KUKA KRL program: Rack_Azul_Abrir_PLC.src, Rack_Azul_Abrir_PLC.dat

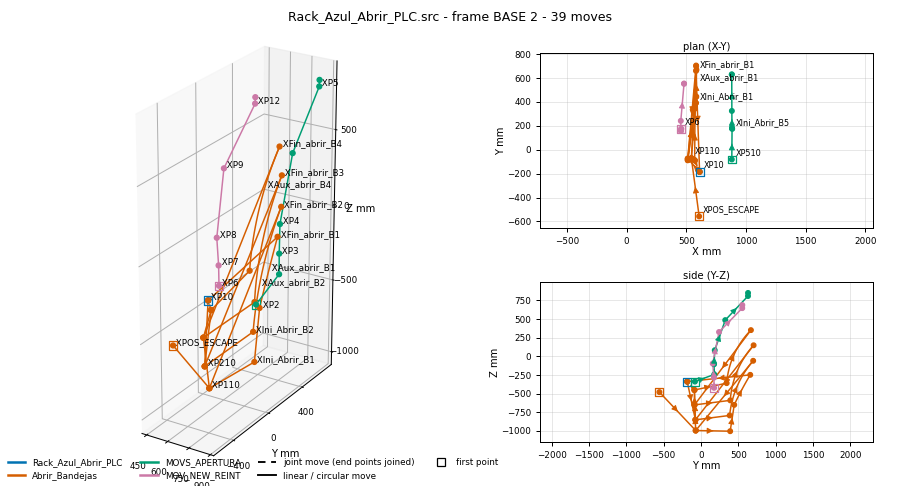
[picture p0: tool path of Rack_Azul_Abrir_PLC.src in frame BASE 2, 39 of 50 moves have a stored position in this frame; points joined in program order, loops and branches not executed]
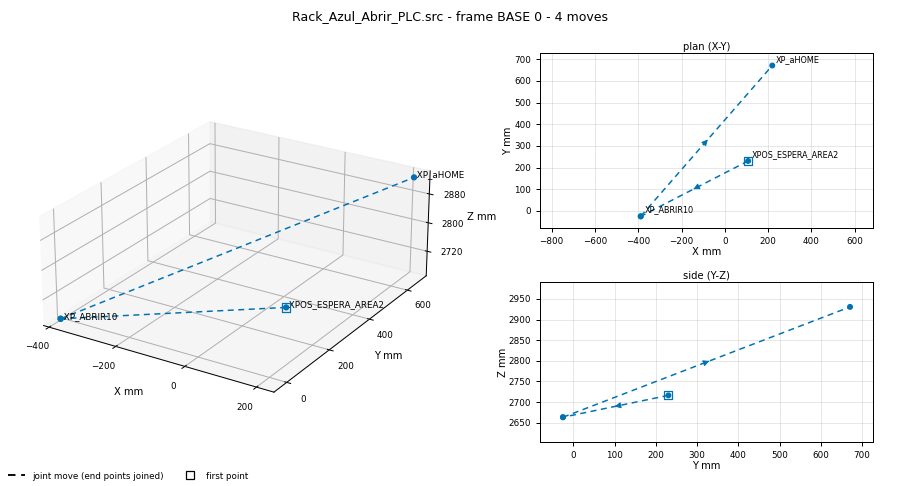
[picture p1: tool path of Rack_Azul_Abrir_PLC.src in frame BASE 0, 4 of 50 moves have a stored position in this frame; points joined in program order, loops and branches not executed]
--- Rack_Azul_Abrir_PLC.src ---
&ACCESS RVO1
&REL 29
&COMMENT ABRIR BAND RACK AZUL
&PARAM EDITMASK = *
&PARAM TEMPLATE = C:\KRC\Roboter\Template\vorgabe
&PARAM DISKPATH = KRC:\R1\Program\MAFELEC
DEF Rack_Azul_Abrir_PLC( )
;FOLD INI;%{PE}
  ;FOLD BASISTECH INI
    GLOBAL INTERRUPT DECL 3 WHEN $STOPMESS==TRUE DO IR_STOPM ( )
    INTERRUPT ON 3
    BAS (#INITMOV,0 )
  ;ENDFOLD (BASISTECH INI)
;FOLD SPOTTECH INI
USERSPOT(#INIT)
;ENDFOLD (SPOTTECH INI)
;FOLD GRIPPERTECH INI
USER_GRP(0,DUMMY,DUMMY,GDEFAULT)
;ENDFOLD (GRIPPERTECH INI)
  ;FOLD USER INI
    ;Make your modifications here
INTERRUPT DECL 21 WHEN I_Rack2_S1 DO Paro()
INTERRUPT DECL 22 WHEN I_Rack2_S2 DO Paro()
INTERRUPT DECL 23 WHEN I_Rack2_S3 DO Paro()
INTERRUPT DECL 24 WHEN I_Rack2_S4 DO Paro()
INTERRUPT DECL 25 WHEN I_Rack2_S5 DO Paro()
INTERRUPT DECL 81 WHEN I_121R1S501 DO STOP_PUSH ()
INTERRUPT DECL 82 WHEN I_121R1S502 DO STOP_PUSH ()
O_TYPE_INFO=0

  ;ENDFOLD (USER INI)
;ENDFOLD (INI)
;################################################
; PROYECTO: MAFELEC PLANTA DE BATERIAS
; ROBOT: 121_R1
; PROGRAMA: APERTURA DE BANDEJAS EN RACK AZUL
; CREADO POR: Su Majestad Felipe VI(zaisor robotics)
; FECHA: 23-NOVIEMBRE-2022
; MODIFICADO POR:
; FECHA MODIFICACION: 18-ENERO-2023
;################################################

Empujador(1,"A",FALSE)
Empujador(2,"R",FALSE)

; POSICION DE ESPERA ENTRADA RACK 2 (AZUL)
;FOLD PTP POS_ESPERA_AREA2 Vel=100 % H Tool[9]:T_Gripper1_Vacio Base[0];%{PE}%R 8.3.48,%MKUKATPBASIS,%CMOVE,%VPTP,%P 1:PTP, 2:POS_ESPERA_AREA2, 3:, 5:100, 7:H
$BWDSTART=FALSE
PDAT_ACT=PH
FDAT_ACT=FPOS_ESPERA_AREA2
BAS(#PTP_PARAMS,100)
PTP XPOS_ESPERA_AREA2
;ENDFOLD

$TIMER[6]=0
$TIMER_STOP[6]=FALSE

;ESPERA AREA 2
WAIT FOR I_ARDY_2
O_AREL_2=FALSE

WAIT FOR I_121R1S1000==FALSE
;INTERRUPT ON 81
;INTERRUPT ON 91

;FOLD PTP P_ABRIR10 CONT Vel=100 % H Tool[9]:T_Gripper1_Vacio Base[0];%{PE}%R 8.3.48,%MKUKATPBASIS,%CMOVE,%VPTP,%P 1:PTP, 2:P_ABRIR10, 3:C_DIS, 5:100, 7:H
$BWDSTART=FALSE
PDAT_ACT=PH
FDAT_ACT=FP_ABRIR10
BAS(#PTP_PARAMS,100)
PTP XP_ABRIR10 C_DIS
;ENDFOLD

;FOLD PTP P10 Vel=100 % H Tool[1]:T_PUSH1 Base[2]:Rack_Azul;%{PE}%R 8.3.48,%MKUKATPBASIS,%CMOVE,%VPTP,%P 1:PTP, 2:P10, 3:, 5:100, 7:H
$BWDSTART=FALSE
PDAT_ACT=PH
FDAT_ACT=FP10
BAS(#PTP_PARAMS,100)
PTP XP10
;ENDFOLD

Empujador(1,"A",TRUE)
Empujador(2,"R",TRUE)

Repite:
Abrir_Bandejas ()

IF INTERRUPT_ACTV THEN
PTP $POS_ACT
GOTO Repite
ENDIF

;FOLD PTP P10 Vel=100 % H Tool[1]:T_PUSH1 Base[2]:Rack_Azul;%{PE}%R 8.3.48,%MKUKATPBASIS,%CMOVE,%VPTP,%P 1:PTP, 2:P10, 3:, 5:100, 7:H
$BWDSTART=FALSE
PDAT_ACT=PH
FDAT_ACT=FP10
BAS(#PTP_PARAMS,100)
PTP XP10
;ENDFOLD

; TRABAJO REALIZADO
O_JRDY_2=TRUE

IF FINALIZA_AZUL==FALSE THEN
O_TYPE_RQ=TRUE
WAIT FOR I_TYPE_INFO==1
ENDIF

O_TYPE_RQ=FALSE

Empujador(1,"R",FALSE)
Empujador(2,"R",FALSE)

; POSICION DE SALIDA RACK 2 (AZUL)
;FOLD PTP POS_AREA2_LIBRE Vel=100 % H Tool[9]:T_Gripper1_Vacio Base[0];%{PE}%R 8.3.48,%MKUKATPBASIS,%CMOVE,%VPTP,%P 1:PTP, 2:POS_AREA2_LIBRE, 3:, 5:100, 7:H
$BWDSTART=FALSE
PDAT_ACT=PH
FDAT_ACT=FPOS_AREA2_LIBRE
BAS(#PTP_PARAMS,100)
PTP XPOS_AREA2_LIBRE
;ENDFOLD
O_AREL_2=TRUE
Empujador(1,"R",TRUE)
Empujador(2,"R",TRUE)

;FOLD PTP P_aHOME CONT Vel=100 % H Tool[9]:T_Gripper1_Vacio Base[0];%{PE}%R 8.3.48,%MKUKATPBASIS,%CMOVE,%VPTP,%P 1:PTP, 2:P_aHOME, 3:C_DIS, 5:100, 7:H
$BWDSTART=FALSE
PDAT_ACT=PH
FDAT_ACT=FP_aHOME
BAS(#PTP_PARAMS,100)
PTP XP_aHOME C_DIS
;ENDFOLD
INTERRUPT OFF 81
INTERRUPT OFF 82

END
DEF Abrir_Bandejas ()

INI_BUCLE:
PTP $POS_ACT
INTERRUPT_ACTV=FALSE

INTERRUPT DECL 86 WHEN I_121R1S501 DO INT_6970 ()
INTERRUPT DECL 87 WHEN I_121R1S502 DO INT_6970 ()
INTERRUPT DECL 88 WHEN I_121R1S501 DO STOP_INT_REINT()
INTERRUPT DECL 89 WHEN I_121R1S502 DO STOP_INT_REINT()
INTERRUPT OFF 86
INTERRUPT OFF 87
INTERRUPT OFF 88
INTERRUPT OFF 89

IF TORQ_HAB THEN
;FOLD TORQMON SetLimits Axis1: 50 % Axis2: 50 % Axis3: 50 % Axis4: 50 % Axis5: 50 % Axis6: 50 %;%{PE}%R 8.3.48,%MKUKATPBASIS,%CTQ_MON,%VTQ_LIMITS,%P 2:TQ_LIMITS, 4:50, 7:50, 10:50, 13:50, 16:50, 19:50
SET_TQ_VALUES (50,50,50,50,50,50)
;ENDFOLD
ENDIF

O_TYPE_RQ=FALSE
WAIT FOR I_TYPE_INFO==0

O_TYPE_RQ=TRUE
WAIT FOR (I_TYPE_INFO > 0) AND (I_TYPE_INFO < 26)
RA_Bandeja_Nr=I_TYPE_INFO
O_TYPE_INFO=I_TYPE_INFO

;PETICION APERTURA BANDEJAS EN RACK 2 (AZUL)
SWITCH RA_Bandeja_Nr ;

CASE 1
O_TYPE_RQ=FALSE
FINALIZA_AZUL=TRUE
;FOLD LIN POS_ESCAPE Vel=1 m/s H Tool[2]:T_PUSH2 Base[2]:Rack_Azul;%{PE}%R 8.3.48,%MKUKATPBASIS,%CMOVE,%VLIN,%P 1:LIN, 2:POS_ESCAPE, 3:, 5:1, 7:H
$BWDSTART=FALSE
LDAT_ACT=LH
FDAT_ACT=FPOS_ESCAPE
BAS(#CP_PARAMS,1)
LIN XPOS_ESCAPE
;ENDFOLD
GOTO FIN

CASE 21
; TRABAJO REALIZADO
O_JRDY_5=FALSE

O_TYPE_RQ=FALSE
FINALIZA_AZUL=FALSE
;FOLD ACTIVA BUSQUEDA APERTURA BANDEJA 1
INTERRUPT ON 21
OLD_OVPRO=$OV_PRO
$ADVANCE=0
;ENDFOLD
WAIT FOR I_Rack2_S2==TRUE
WAIT FOR I_Rack2_S1==FALSE

WAIT FOR I_RackAzul_Pin2A
WAIT FOR I_RackAzul_Pin1B

;FOLD LIN P110 CONT Vel=1 m/s M Tool[1]:T_PUSH1 Base[2]:Rack_Azul;%{PE}%R 8.3.48,%MKUKATPBASIS,%CMOVE,%VLIN,%P 1:LIN, 2:P110, 3:C_DIS C_DIS, 5:1, 7:M
$BWDSTART=FALSE
LDAT_ACT=LM
FDAT_ACT=FP110
BAS(#CP_PARAMS,1)
LIN XP110 C_DIS C_DIS
;ENDFOLD

;FOLD LIN Ini_Abrir_B1 Vel=1 m/s M Tool[1]:T_PUSH1 Base[2]:Rack_Azul;%{PE}%R 8.3.48,%MKUKATPBASIS,%CMOVE,%VLIN,%P 1:LIN, 2:Ini_Abrir_B1, 3:, 5:1, 7:M
$BWDSTART=FALSE
LDAT_ACT=LM
FDAT_ACT=FIni_Abrir_B1
BAS(#CP_PARAMS,1)
LIN XIni_Abrir_B1
;ENDFOLD
;FOLD LIN P2 CONT Vel=1 m/s M Tool[1]:T_PUSH1 Base[2]:Rack_Azul;%{PE}%R 8.3.48,%MKUKATPBASIS,%CMOVE,%VLIN,%P 1:LIN, 2:P2, 3:C_DIS C_DIS, 5:1, 7:M
$BWDSTART=FALSE
LDAT_ACT=LM
FDAT_ACT=FP2
BAS(#CP_PARAMS,1)
LIN XP2 C_DIS C_DIS
;ENDFOLD
;FOLD CIRC Aux_abrir_B1 Fin_abrir_B1 CONT Vel=1 m/s M Tool[1]:T_PUSH1 Base[2]:Rack_Azul;%{PE}%R 8.3.48,%MKUKATPBASIS,%CMOVE,%VCIRC,%P 1:CIRC, 2:Aux_abrir_B1, 3:Fin_abrir_B1, 4:C_DIS C_DIS, 6:1, 8:M
$BWDSTART=FALSE
LDAT_ACT=LM
FDAT_ACT=FFin_abrir_B1
BAS(#CP_PARAMS,1)
CIRC XAux_abrir_B1, XFin_abrir_B1 C_DIS C_DIS
;ENDFOLD
LIN_REL{y 5}
LIN_REL{Z 10}
O_TREQ_3=TRUE
WAIT FOR I_TRDY_3
O_TREQ_3=FALSE

; TRABAJO REALIZADO
O_JRDY_5=TRUE

;FOLD LIN P120 CONT Vel=1 m/s M Tool[1]:T_PUSH1 Base[2]:Rack_Azul;%{PE}%R 8.3.48,%MKUKATPBASIS,%CMOVE,%VLIN,%P 1:LIN, 2:P120, 3:C_DIS C_DIS, 5:1, 7:M
$BWDSTART=FALSE
LDAT_ACT=LM
FDAT_ACT=FP120
BAS(#CP_PARAMS,1)
LIN XP120 C_DIS C_DIS
;ENDFOLD
GOTO FIN

CASE 22
; TRABAJO REALIZADO
O_JRDY_5=FALSE

O_TYPE_RQ=FALSE
FINALIZA_AZUL=FALSE
;FOLD ACTIVA BUSQUEDA APERTURA BANDEJA 2
INTERRUPT ON 22
OLD_OVPRO=$OV_PRO
$ADVANCE=0
;ENDFOLD
WAIT FOR I_Rack2_S3==TRUE
WAIT FOR I_Rack2_S2==FALSE

WAIT FOR I_RackAzul_Pin3A
WAIT FOR I_RackAzul_Pin2B

;FOLD LIN P210 CONT Vel=1 m/s M Tool[1]:T_PUSH1 Base[2]:Rack_Azul;%{PE}%R 8.3.48,%MKUKATPBASIS,%CMOVE,%VLIN,%P 1:LIN, 2:P210, 3:C_DIS C_DIS, 5:1, 7:M
$BWDSTART=FALSE
LDAT_ACT=LM
FDAT_ACT=FP210
BAS(#CP_PARAMS,1)
LIN XP210 C_DIS C_DIS
;ENDFOLD
;FOLD LIN Ini_Abrir_B2 Vel=1 m/s M Tool[1]:T_PUSH1 Base[2]:Rack_Azul;%{PE}%R 8.3.48,%MKUKATPBASIS,%CMOVE,%VLIN,%P 1:LIN, 2:Ini_Abrir_B2, 3:, 5:1, 7:M
$BWDSTART=FALSE
LDAT_ACT=LM
FDAT_ACT=FIni_Abrir_B2
BAS(#CP_PARAMS,1)
LIN XIni_Abrir_B2
;ENDFOLD
;FOLD CIRC Aux_abrir_B2 Fin_abrir_B2 CONT Vel=1 m/s M Tool[1]:T_PUSH1 Base[2]:Rack_Azul;%{PE}%R 8.3.48,%MKUKATPBASIS,%CMOVE,%VCIRC,%P 1:CIRC, 2:Aux_abrir_B2, 3:Fin_abrir_B2, 4:C_DIS C_DIS, 6:1, 8:M
$BWDSTART=FALSE
LDAT_ACT=LM
FDAT_ACT=FFin_abrir_B2
BAS(#CP_PARAMS,1)
CIRC XAux_abrir_B2, XFin_abrir_B2 C_DIS C_DIS
;ENDFOLD
LIN_REL{Z 10}
O_TREQ_3=TRUE
WAIT FOR I_TRDY_3
O_TREQ_3=FALSE

; TRABAJO REALIZADO
O_JRDY_5=TRUE

;FOLD LIN P220 CONT Vel=1 m/s M Tool[1]:T_PUSH1 Base[2]:Rack_Azul;%{PE}%R 8.3.48,%MKUKATPBASIS,%CMOVE,%VLIN,%P 1:LIN, 2:P220, 3:C_DIS C_DIS, 5:1, 7:M
$BWDSTART=FALSE
LDAT_ACT=LM
FDAT_ACT=FP220
BAS(#CP_PARAMS,1)
LIN XP220 C_DIS C_DIS
;ENDFOLD
;FOLD LIN P110 CONT Vel=1 m/s M Tool[1]:T_PUSH1 Base[2]:Rack_Azul;%{PE}%R 8.3.48,%MKUKATPBASIS,%CMOVE,%VLIN,%P 1:LIN, 2:P110, 3:C_DIS C_DIS, 5:1, 7:M
$BWDSTART=FALSE
LDAT_ACT=LM
FDAT_ACT=FP110
BAS(#CP_PARAMS,1)
LIN XP110 C_DIS C_DIS
;ENDFOLD
GOTO INI_BUCLE

CASE 23
; TRABAJO REALIZADO
O_JRDY_5=FALSE

O_TYPE_RQ=FALSE
FINALIZA_AZUL=FALSE
;FOLD ACTIVA BUSQUEDA APERTURA BANDEJA 3
INTERRUPT ON 23
OLD_OVPRO=$OV_PRO
$ADVANCE=0
;ENDFOLD
WAIT FOR I_Rack2_S4==TRUE
WAIT FOR I_Rack2_S3==FALSE

WAIT FOR I_RackAzul_Pin4A
WAIT FOR I_RackAzul_Pin3B

;FOLD LIN P310 CONT Vel=1 m/s M Tool[1]:T_PUSH1 Base[2]:Rack_Azul;%{PE}%R 8.3.48,%MKUKATPBASIS,%CMOVE,%VLIN,%P 1:LIN, 2:P310, 3:C_DIS C_DIS, 5:1, 7:M
$BWDSTART=FALSE
LDAT_ACT=LM
FDAT_ACT=FP310
BAS(#CP_PARAMS,1)
LIN XP310 C_DIS C_DIS
;ENDFOLD
;FOLD LIN Ini_Abrir_B3 Vel=1 m/s M Tool[1]:T_PUSH1 Base[2]:Rack_Azul;%{PE}%R 8.3.48,%MKUKATPBASIS,%CMOVE,%VLIN,%P 1:LIN, 2:Ini_Abrir_B3, 3:, 5:1, 7:M
$BWDSTART=FALSE
LDAT_ACT=LM
FDAT_ACT=FIni_Abrir_B3
BAS(#CP_PARAMS,1)
LIN XIni_Abrir_B3
;ENDFOLD
;FOLD CIRC Aux_abrir_B3 Fin_abrir_B3 CONT Vel=1 m/s M Tool[1]:T_PUSH1 Base[2]:Rack_Azul;%{PE}%R 8.3.48,%MKUKATPBASIS,%CMOVE,%VCIRC,%P 1:CIRC, 2:Aux_abrir_B3, 3:Fin_abrir_B3, 4:C_DIS C_DIS, 6:1, 8:M
$BWDSTART=FALSE
LDAT_ACT=LM
FDAT_ACT=FFin_abrir_B3
BAS(#CP_PARAMS,1)
CIRC XAux_abrir_B3, XFin_abrir_B3 C_DIS C_DIS
;ENDFOLD
LIN_REL{Z 10}
O_TREQ_3=TRUE
WAIT FOR I_TRDY_3
O_TREQ_3=FALSE

; TRABAJO REALIZADO
O_JRDY_5=TRUE

;FOLD LIN P320 CONT Vel=1 m/s M Tool[1]:T_PUSH1 Base[2]:Rack_Azul;%{PE}%R 8.3.48,%MKUKATPBASIS,%CMOVE,%VLIN,%P 1:LIN, 2:P320, 3:C_DIS C_DIS, 5:1, 7:M
$BWDSTART=FALSE
LDAT_ACT=LM
FDAT_ACT=FP320
BAS(#CP_PARAMS,1)
LIN XP320 C_DIS C_DIS
;ENDFOLD
;FOLD LIN P210 CONT Vel=1 m/s M Tool[1]:T_PUSH1 Base[2]:Rack_Azul;%{PE}%R 8.3.48,%MKUKATPBASIS,%CMOVE,%VLIN,%P 1:LIN, 2:P210, 3:C_DIS C_DIS, 5:1, 7:M
$BWDSTART=FALSE
LDAT_ACT=LM
FDAT_ACT=FP210
BAS(#CP_PARAMS,1)
LIN XP210 C_DIS C_DIS
;ENDFOLD
GOTO INI_BUCLE

CASE 24
; TRABAJO REALIZADO
O_JRDY_5=FALSE

O_TYPE_RQ=FALSE
FINALIZA_VERDE=FALSE
;FOLD ACTIVA BUSQUEDA APERTURA BANDEJA 4
INTERRUPT ON 24
OLD_OVPRO=$OV_PRO
$ADVANCE=0
;ENDFOLD
WAIT FOR I_Rack2_S5==TRUE
WAIT FOR I_Rack2_S4==FALSE

WAIT FOR I_RackAzul_Pin5A
WAIT FOR I_RackAzul_Pin4B

;FOLD LIN P410 CONT Vel=1 m/s M Tool[1]:T_PUSH1 Base[2]:Rack_Azul;%{PE}%R 8.3.48,%MKUKATPBASIS,%CMOVE,%VLIN,%P 1:LIN, 2:P410, 3:C_DIS C_DIS, 5:1, 7:M
$BWDSTART=FALSE
LDAT_ACT=LM
FDAT_ACT=FP410
BAS(#CP_PARAMS,1)
LIN XP410 C_DIS C_DIS
;ENDFOLD
;FOLD LIN Ini_Abrir_B4 Vel=1 m/s M Tool[1]:T_PUSH1 Base[2]:Rack_Azul;%{PE}%R 8.3.48,%MKUKATPBASIS,%CMOVE,%VLIN,%P 1:LIN, 2:Ini_Abrir_B4, 3:, 5:1, 7:M
$BWDSTART=FALSE
LDAT_ACT=LM
FDAT_ACT=FIni_Abrir_B4
BAS(#CP_PARAMS,1)
LIN XIni_Abrir_B4
;ENDFOLD
;FOLD CIRC Aux_abrir_B4 Fin_abrir_B4 CONT Vel=1 m/s M Tool[1]:T_PUSH1 Base[2]:Rack_Azul;%{PE}%R 8.3.48,%MKUKATPBASIS,%CMOVE,%VCIRC,%P 1:CIRC, 2:Aux_abrir_B4, 3:Fin_abrir_B4, 4:C_DIS C_DIS, 6:1, 8:M
$BWDSTART=FALSE
LDAT_ACT=LM
FDAT_ACT=FFin_abrir_B4
BAS(#CP_PARAMS,1)
CIRC XAux_abrir_B4, XFin_abrir_B4 C_DIS C_DIS
;ENDFOLD
LIN_REL{Z 10}
O_TREQ_3=TRUE
WAIT FOR I_TRDY_3
O_TREQ_3=FALSE

; TRABAJO REALIZADO
O_JRDY_5=TRUE

;FOLD LIN P420 CONT Vel=1 m/s M Tool[1]:T_PUSH1 Base[2]:Rack_Azul;%{PE}%R 8.3.48,%MKUKATPBASIS,%CMOVE,%VLIN,%P 1:LIN, 2:P420, 3:C_DIS C_DIS, 5:1, 7:M
$BWDSTART=FALSE
LDAT_ACT=LM
FDAT_ACT=FP420
BAS(#CP_PARAMS,1)
LIN XP420 C_DIS C_DIS
;ENDFOLD
;FOLD LIN P310 CONT Vel=1 m/s M Tool[1]:T_PUSH1 Base[2]:Rack_Azul;%{PE}%R 8.3.48,%MKUKATPBASIS,%CMOVE,%VLIN,%P 1:LIN, 2:P310, 3:C_DIS C_DIS, 5:1, 7:M
$BWDSTART=FALSE
LDAT_ACT=LM
FDAT_ACT=FP310
BAS(#CP_PARAMS,1)
LIN XP310 C_DIS C_DIS
;ENDFOLD
GOTO INI_BUCLE

CASE 25

INTERRUPT ON 81
INTERRUPT ON 82


; TRABAJO REALIZADO
O_JRDY_5=FALSE

O_TYPE_RQ=FALSE
FINALIZA_AZUL=FALSE
;FOLD ACTIVA BUSQUEDA APERTURA BANDEJA 5
INTERRUPT ON 25
OLD_OVPRO=$OV_PRO
$ADVANCE=0
;ENDFOLD
WAIT FOR I_Rack2_S5==FALSE
WAIT FOR I_RackAzul_Pin5B

$advance=2

MOVS_APERTURA()
IF REINT_APERTURA==TRUE THEN
   MOV_NEW_REINT()
ENDIF


$advance=0
O_TREQ_3=TRUE
WAIT FOR I_TRDY_3
O_TREQ_3=FALSE

; TRABAJO REALIZADO
O_JRDY_5=TRUE

;FOLD LIN P520 CONT Vel=1 m/s M Tool[1]:T_PUSH1 Base[2]:Rack_Azul;%{PE}%R 8.3.48,%MKUKATPBASIS,%CMOVE,%VLIN,%P 1:LIN, 2:P520, 3:C_DIS C_DIS, 5:1, 7:M
$BWDSTART=FALSE
LDAT_ACT=LM
FDAT_ACT=FP520
BAS(#CP_PARAMS,1)
LIN XP520 C_DIS C_DIS
;ENDFOLD
;FOLD LIN P410 CONT Vel=1 m/s H Tool[1]:T_PUSH1 Base[2]:Rack_Azul;%{PE}%R 8.3.48,%MKUKATPBASIS,%CMOVE,%VLIN,%P 1:LIN, 2:P410, 3:C_DIS C_DIS, 5:1, 7:H
$BWDSTART=FALSE
LDAT_ACT=LH
FDAT_ACT=FP410
BAS(#CP_PARAMS,1)
LIN XP410 C_DIS C_DIS
;ENDFOLD
GOTO INI_BUCLE

DEFAULT
HALT
HALT
HALT
ENDSWITCH

FIN:

;FOLD TORQMON SetDefault;%{PE}%R 8.3.48,%MKUKATPBASIS,%CTQ_MON,%VTQ_DEFAULT,%P 2:TQ_DEFAULT
SET_TQ_VALUES ( )
;ENDFOLD

;FOLD PTP P10 CONT Vel=100 % H Tool[1]:T_PUSH1 Base[2]:Rack_Azul;%{PE}%R 8.3.48,%MKUKATPBASIS,%CMOVE,%VPTP,%P 1:PTP, 2:P10, 3:C_DIS, 5:100, 7:H
$BWDSTART=FALSE
PDAT_ACT=PH
FDAT_ACT=FP10
BAS(#PTP_PARAMS,100)
PTP XP10 C_DIS
;ENDFOLD

$TIMER_STOP[6]=TRUE
END
DEF Paro()
INTERRUPT OFF 21
INTERRUPT OFF 22
INTERRUPT OFF 23
INTERRUPT OFF 24
INTERRUPT OFF 25

IF I_Rack2_S1 THEN
INTERRUPT_ACTV=FALSE
ELSE
INTERRUPT_ACTV=TRUE
ENDIF

BRAKE

WAIT SEC 0

PTP $POS_ACT
LIN $POS_INT

$OV_PRO=OLD_OVPRO

O_TREQ_3=TRUE
WAIT FOR I_TRDY_3
O_TREQ_3=FALSE

; TRABAJO REALIZADO
O_JRDY_5=TRUE

RESUME

END
DEF STOP_PUSH ()
INTERRUPT OFF 81
INTERRUPT OFF 82
BRAKE
PTP $POS_ACT
LIN_REL{Z -50}
WAIT SEC 0.5
WAIT FOR (NOT I_121R1S501) AND (NOT I_121R1S502)
LIN_REL{Z 50}
PTP $POS_ACT
;RESUME
END
DEF MOVS_APERTURA()
REINT_APERTURA=FALSE
INTERRUPT OFF 81
INTERRUPT OFF 82
INTERRUPT ON 86
INTERRUPT ON 87


;FOLD LIN P510 CONT Vel=0.5 m/s M Tool[1]:T_PUSH1 Base[2]:Rack_Azul;%{PE}%R 8.3.48,%MKUKATPBASIS,%CMOVE,%VLIN,%P 1:LIN, 2:P510, 3:C_DIS C_DIS, 5:0.5, 7:M
$BWDSTART=FALSE
LDAT_ACT=LM
FDAT_ACT=FP510
BAS(#CP_PARAMS,0.5)
LIN XP510 C_DIS C_DIS
;ENDFOLD
;FOLD LIN Ini_Abrir_B5 Vel=0.5 m/s M Tool[1]:T_PUSH1 Base[2]:Rack_Azul;%{PE}%R 8.3.48,%MKUKATPBASIS,%CMOVE,%VLIN,%P 1:LIN, 2:Ini_Abrir_B5, 3:, 5:0.5, 7:M
$BWDSTART=FALSE
LDAT_ACT=LM
FDAT_ACT=FIni_Abrir_B5
BAS(#CP_PARAMS,0.5)
LIN XIni_Abrir_B5
;ENDFOLD

;FOLD LIN P3 CONT Vel=0.1 m/s M2 Tool[1]:T_PUSH1 Base[2]:Rack_Azul;%{PE}%R 8.3.48,%MKUKATPBASIS,%CMOVE,%VLIN,%P 1:LIN, 2:P3, 3:C_DIS C_DIS, 5:0.1, 7:M2
$BWDSTART=FALSE
LDAT_ACT=LM2
FDAT_ACT=FP3
BAS(#CP_PARAMS,0.1)
LIN XP3 C_DIS C_DIS
;ENDFOLD
;FOLD LIN P4 CONT Vel=0.1 m/s M2 Tool[1]:T_PUSH1 Base[2]:Rack_Azul;%{PE}%R 8.3.48,%MKUKATPBASIS,%CMOVE,%VLIN,%P 1:LIN, 2:P4, 3:C_DIS C_DIS, 5:0.1, 7:M2
$BWDSTART=FALSE
LDAT_ACT=LM2
FDAT_ACT=FP4
BAS(#CP_PARAMS,0.1)
LIN XP4 C_DIS C_DIS
;ENDFOLD
;FOLD LIN Aux_abrir_B5 CONT Vel=1 m/s M2 Tool[1]:T_PUSH1 Base[2]:Rack_Azul;%{PE}%R 8.3.48,%MKUKATPBASIS,%CMOVE,%VLIN,%P 1:LIN, 2:Aux_abrir_B5, 3:C_DIS C_DIS, 5:1, 7:M2
$BWDSTART=FALSE
LDAT_ACT=LM2
FDAT_ACT=FAux_abrir_B5
BAS(#CP_PARAMS,1)
LIN XAux_abrir_B5 C_DIS C_DIS
;ENDFOLD
;FOLD LIN P5 CONT Vel=1 m/s M2 Tool[1]:T_PUSH1 Base[2]:Rack_Azul;%{PE}%R 8.3.48,%MKUKATPBASIS,%CMOVE,%VLIN,%P 1:LIN, 2:P5, 3:C_DIS C_DIS, 5:1, 7:M2
$BWDSTART=FALSE
LDAT_ACT=LM2
FDAT_ACT=FP5
BAS(#CP_PARAMS,1)
LIN XP5 C_DIS C_DIS
;ENDFOLD
;FOLD LIN Fin_abrir_B5 CONT Vel=1 m/s M2 Tool[1]:T_PUSH1 Base[2]:Rack_Azul;%{PE}%R 8.3.48,%MKUKATPBASIS,%CMOVE,%VLIN,%P 1:LIN, 2:Fin_abrir_B5, 3:C_DIS C_DIS, 5:1, 7:M2
$BWDSTART=FALSE
LDAT_ACT=LM2
FDAT_ACT=FFin_abrir_B5
BAS(#CP_PARAMS,1)
LIN XFin_abrir_B5 C_DIS C_DIS
;ENDFOLD

END
DEF INT_6970()

BRAKE
INTERRUPT OFF 86
INTERRUPT OFF 87
REINT_APERTURA=TRUE
RESUME

END
DEF MOV_NEW_REINT()

INTERRUPT ON 88
INTERRUPT ON 89


;FOLD LIN P6 CONT Vel=0.5 m/s CPDAT2 Tool[2]:T_PUSH2 Base[2]:Rack_Azul;%{PE}%R 8.3.48,%MKUKATPBASIS,%CMOVE,%VLIN,%P 1:LIN, 2:P6, 3:C_DIS C_DIS, 5:0.5, 7:CPDAT2
$BWDSTART=FALSE
LDAT_ACT=LCPDAT2
FDAT_ACT=FP6
BAS(#CP_PARAMS,0.5)
LIN XP6 C_DIS C_DIS
;ENDFOLD
;FOLD LIN P7 CONT Vel=0.1 m/s CPDAT3 Tool[2]:T_PUSH2 Base[2]:Rack_Azul;%{PE}%R 8.3.48,%MKUKATPBASIS,%CMOVE,%VLIN,%P 1:LIN, 2:P7, 3:C_DIS C_DIS, 5:0.1, 7:CPDAT3
$BWDSTART=FALSE
LDAT_ACT=LCPDAT3
FDAT_ACT=FP7
BAS(#CP_PARAMS,0.1)
LIN XP7 C_DIS C_DIS
;ENDFOLD
;FOLD LIN P8 CONT Vel=0.1 m/s CPDAT4 Tool[2]:T_PUSH2 Base[2]:Rack_Azul;%{PE}%R 8.3.48,%MKUKATPBASIS,%CMOVE,%VLIN,%P 1:LIN, 2:P8, 3:C_DIS C_DIS, 5:0.1, 7:CPDAT4
$BWDSTART=FALSE
LDAT_ACT=LCPDAT4
FDAT_ACT=FP8
BAS(#CP_PARAMS,0.1)
LIN XP8 C_DIS C_DIS
;ENDFOLD
;FOLD LIN P9 CONT Vel=0.1 m/s CPDAT5 Tool[2]:T_PUSH2 Base[2]:Rack_Azul;%{PE}%R 8.3.48,%MKUKATPBASIS,%CMOVE,%VLIN,%P 1:LIN, 2:P9, 3:C_DIS C_DIS, 5:0.1, 7:CPDAT5
$BWDSTART=FALSE
LDAT_ACT=LCPDAT5
FDAT_ACT=FP9
BAS(#CP_PARAMS,0.1)
LIN XP9 C_DIS C_DIS
;ENDFOLD
;FOLD LIN P12 CONT Vel=0.1 m/s CPDAT6 Tool[2]:T_PUSH2 Base[2]:Rack_Azul;%{PE}%R 8.3.48,%MKUKATPBASIS,%CMOVE,%VLIN,%P 1:LIN, 2:P12, 3:C_DIS C_DIS, 5:0.1, 7:CPDAT6
$BWDSTART=FALSE
LDAT_ACT=LCPDAT6
FDAT_ACT=FP12
BAS(#CP_PARAMS,0.1)
LIN XP12 C_DIS C_DIS
;ENDFOLD
;FOLD LIN P13 CONT Vel=0.1 m/s CPDAT7 Tool[2]:T_PUSH2 Base[2]:Rack_Azul;%{PE}%R 8.3.48,%MKUKATPBASIS,%CMOVE,%VLIN,%P 1:LIN, 2:P13, 3:C_DIS C_DIS, 5:0.1, 7:CPDAT7
$BWDSTART=FALSE
LDAT_ACT=LCPDAT7
FDAT_ACT=FP13
BAS(#CP_PARAMS,0.1)
LIN XP13 C_DIS C_DIS
;ENDFOLD

END
DEF STOP_INT_REINT()

BRAKE
INTERRUPT OFF 88
INTERRUPT OFF 89
WAIT FOR FALSE
;2DO REINTENTO APERTURA FALLIDO
;ABRIR BANDEJA A MANO
;SELECCIONAR PASO AQUI Y LEER EL PTP DE LA LINEA SIGUIENTE
PTP $POS_ACT

END

--- Rack_Azul_Abrir_PLC.dat ---
&ACCESS RVO1
&REL 29
&COMMENT ABRIR BAND RACK AZUL
&PARAM EDITMASK = *
&PARAM TEMPLATE = C:\KRC\Roboter\Template\vorgabe
&PARAM DISKPATH = KRC:\R1\Program\MAFELEC
DEFDAT  Rack_Azul_Abrir_PLC
;FOLD EXTERNAL DECLARATIONS;%{PE}%MKUKATPBASIS,%CEXT,%VCOMMON,%P
;FOLD GRIPPERTECH EXT
EXT  H50 (INT  :IN,INT  :IN,INT  :IN,GRP_TYP  :IN )
;ENDFOLD (GRIPPERTECH EXT)
;FOLD SPOTTECH EXT
EXT  USERSPOT (S_COMMAND  :IN,SPOT_TYPE  :IN )
;ENDFOLD (SPOTTECH EXT)
;FOLD BASISTECH EXT;%{PE}%MKUKATPBASIS,%CEXT,%VEXT,%P
EXT  BAS (BAS_COMMAND  :IN,REAL  :IN )
DECL INT SUCCESS
;ENDFOLD (BASISTECH EXT)
;FOLD USER EXT;%{E}%MKUKATPUSER,%CEXT,%VEXT,%P
;Make your modifications here

;ENDFOLD (USER EXT)
;ENDFOLD (EXTERNAL DECLARATIONS)
DECL BASIS_SUGG_T LAST_BASIS={POINT1[] "P13                     ",POINT2[] "P13                     ",CP_PARAMS[] "CPDAT7                  ",PTP_PARAMS[] "PDAT0                   ",CONT[] "C_DIS C_DIS             ",CP_VEL[] "0.1                     ",PTP_VEL[] " 100                    ",SYNC_PARAMS[] "SYNCDAT                 ",SPL_NAME[] "S0                      ",A_PARAMS[] "ADAT0                   "}
DECL PDAT PH={VEL 100.000,ACC 100.000,APO_DIST 100.000,APO_MODE #CDIS,GEAR_JERK 50.0000,EXAX_IGN 0}
DECL E6POS XPOS_ESPERA_AREA1={X 112.943756,Y -227.851166,Z 2716.11304,A 36.2463837,B -15.5853510,C 56.0520973,S 3,T 42,E1 0.0,E2 0.0,E3 0.0,E4 0.0,E5 0.0,E6 0.0}
DECL FDAT FPOS_ESPERA_AREA1={TOOL_NO 9,BASE_NO 0,IPO_FRAME #BASE,POINT2[] " ",TQ_STATE FALSE}
DECL E6POS XAUX_ABRIR_B1={X 583.925598,Y 553.971619,Z -433.916260,A 89.1835861,B 28.1399021,C -90.0818,S 6,T 19,E1 0.0,E2 0.0,E3 0.0,E4 0.0,E5 0.0,E6 0.0}
DECL E6POS XFIN_ABRIR_B1={X 581.448059,Y 660.397583,Z -247.272278,A 90.1830063,B 16.3026943,C -89.0826797,S 6,T 19,E1 0.0,E2 0.0,E3 0.0,E4 0.0,E5 0.0,E6 0.0}
DECL FDAT FFin_abrir_B1={TOOL_NO 1,BASE_NO 2,IPO_FRAME #BASE,POINT2[] "XAux_abrir_B1",TQ_STATE FALSE}
DECL LDAT LL={VEL 2.00000,ACC 25.0000,APO_DIST 25.0000,APO_FAC 50.0000,AXIS_VEL 100.000,AXIS_ACC 100.000,ORI_TYP #VAR,CIRC_TYP #BASE,JERK_FAC 50.0000,GEAR_JERK 50.0000,EXAX_IGN 0}
DECL E6POS XIni_Abrir_B1={X 580.733337,Y 391.137238,Z -1002.73444,A 88.0927277,B 38.9319153,C -91.1217651,S 6,T 19,E1 0.0,E2 0.0,E3 0.0,E4 0.0,E5 0.0,E6 0.0}
DECL FDAT FIni_Abrir_B1={TOOL_NO 1,BASE_NO 2,IPO_FRAME #BASE,POINT2[] " ",TQ_STATE FALSE}
DECL E6POS XIni_Abrir_B2={X 575.186035,Y 384.262360,Z -791.443298,A 88.1378555,B 31.1529427,C -90.2718658,S 6,T 19,E1 0.0,E2 0.0,E3 0.0,E4 0.0,E5 0.0,E6 0.0}
DECL FDAT FIni_Abrir_B2={TOOL_NO 1,BASE_NO 2,IPO_FRAME #BASE,POINT2[] " ",TQ_STATE FALSE}
DECL E6POS XIni_Abrir_B3={X 579.486511,Y 392.628723,Z -589.202393,A 89.2266464,B 31.1225376,C -89.9745331,S 6,T 19,E1 0.0,E2 0.0,E3 0.0,E4 0.0,E5 0.0,E6 0.0}
DECL FDAT FIni_Abrir_B3={TOOL_NO 1,BASE_NO 2,IPO_FRAME #BASE,POINT2[] " ",TQ_STATE FALSE}
DECL E6POS XIni_Abrir_B4={X 573.262207,Y 344.347107,Z -358.451721,A 89.3433304,B 32.7624969,C -89.6608429,S 6,T 19,E1 0.0,E2 0.0,E3 0.0,E4 0.0,E5 0.0,E6 0.0}
DECL FDAT FIni_Abrir_B4={TOOL_NO 1,BASE_NO 2,IPO_FRAME #BASE,POINT2[] " ",TQ_STATE FALSE}
DECL E6POS XIni_Abrir_B5={X 883.313538,Y 177.747177,Z -241.618011,A 87.2811890,B 0.879289,C -89.4738693,S 6,T 19,E1 0.0,E2 0.0,E3 0.0,E4 0.0,E5 0.0,E6 0.0}
DECL FDAT FIni_Abrir_B5={TOOL_NO 1,BASE_NO 2,IPO_FRAME #BASE,POINT2[] " ",TQ_STATE FALSE}
DECL E6POS XAux_abrir_B2={X 580.652710,Y 447.795807,Z -496.778870,A 88.1063766,B 26.1448574,C -90.1987457,S 6,T 19,E1 0.0,E2 0.0,E3 0.0,E4 0.0,E5 0.0,E6 0.0}
DECL E6POS XFin_abrir_B2={X 582.748474,Y 699.544312,Z -58.7800102,A 88.0612335,B 18.1576080,C -90.0750961,S 6,T 19,E1 0.0,E2 0.0,E3 0.0,E4 0.0,E5 0.0,E6 0.0}
DECL FDAT FFin_abrir_B2={TOOL_NO 1,BASE_NO 2,IPO_FRAME #BASE,POINT2[] "XAux_abrir_B2",TQ_STATE FALSE}
DECL E6POS XAux_abrir_B3={X 582.726868,Y 481.624420,Z -205.312073,A 89.2074585,B 21.3034344,C -89.7415237,S 6,T 19,E1 0.0,E2 0.0,E3 0.0,E4 0.0,E5 0.0,E6 0.0}
DECL E6POS XFin_abrir_B3={X 582.122864,Y 705.353943,Z 149.093140,A 89.1909790,B 11.6588039,C -89.5089874,S 6,T 19,E1 0.0,E2 0.0,E3 0.0,E4 0.0,E5 0.0,E6 0.0}
DECL FDAT FFin_abrir_B3={TOOL_NO 1,BASE_NO 2,IPO_FRAME #BASE,POINT2[] "XAux_abrir_B3",TQ_STATE FALSE}
DECL E6POS XAux_abrir_B4={X 582.759338,Y 506.277557,Z 143.456680,A 90.6976166,B 19.7625904,C -89.0678711,S 6,T 19,E1 0.0,E2 0.0,E3 0.0,E4 0.0,E5 0.0,E6 0.0}
DECL E6POS XFin_abrir_B4={X 585.431213,Y 669.141296,Z 352.292206,A 91.3099213,B 12.9905615,C -88.9002304,S 6,T 19,E1 0.0,E2 0.0,E3 0.0,E4 0.0,E5 0.0,E6 0.0}
DECL FDAT FFin_abrir_B4={TOOL_NO 1,BASE_NO 2,IPO_FRAME #BASE,POINT2[] "XAux_abrir_B4",TQ_STATE FALSE}
DECL E6POS XAux_abrir_B5={X 881.577148,Y 325.192474,Z 486.332092,A 90.6172867,B 27.5276222,C -88.2672195,S 6,T 51,E1 0.0,E2 0.0,E3 0.0,E4 0.0,E5 0.0,E6 0.0}
DECL E6POS XFin_abrir_B5={X 881.470825,Y 630.741699,Z 850.776123,A 92.3442612,B 25.1508522,C -87.7190857,S 6,T 51,E1 0.0,E2 0.0,E3 0.0,E4 0.0,E5 0.0,E6 0.0}
DECL FDAT FFin_abrir_B5={TOOL_NO 1,BASE_NO 2,IPO_FRAME #BASE,POINT2[] " ",TQ_STATE FALSE}
DECL E6POS XPOS_AREA1_LIBRE={X -250.533554,Y -43.6507149,Z 2716.11304,A -84.6604385,B 6.50295877,C 57.2217522,S 3,T 42,E1 0.0,E2 0.0,E3 0.0,E4 0.0,E5 0.0,E6 0.0}
DECL FDAT FPOS_AREA1_LIBRE={TOOL_NO 9,BASE_NO 0,IPO_FRAME #BASE,POINT2[] " ",TQ_STATE FALSE}
DECL E6POS XP111={X -1283.23694,Y -1560.93347,Z 479.113342,A -88.4105606,B 32.4816132,C 90.4043961,S 6,T 58,E1 0.0,E2 0.0,E3 0.0,E4 0.0,E5 0.0,E6 0.0}
DECL FDAT FP111={TOOL_NO 1,BASE_NO 2,IPO_FRAME #BASE,POINT2[] " ",TQ_STATE FALSE}
DECL E6POS XP510={X 881.106140,Y -81.2473831,Z -337.977234,A 89.7929459,B 38.2149963,C -89.0848160,S 6,T 19,E1 0.0,E2 0.0,E3 0.0,E4 0.0,E5 0.0,E6 0.0}
DECL FDAT FP510={TOOL_NO 1,BASE_NO 2,IPO_FRAME #BASE,POINT2[] " ",TQ_STATE FALSE}
DECL E6POS XP520={X 570.135315,Y -87.9825745,Z -450.345490,A 87.9885483,B 38.2075691,C -88.4547653,S 6,T 19,E1 0.0,E2 0.0,E3 0.0,E4 0.0,E5 0.0,E6 0.0}
DECL FDAT FP520={TOOL_NO 1,BASE_NO 2,IPO_FRAME #BASE,POINT2[] " ",TQ_STATE FALSE}
DECL E6POS XP10={X 611.491699,Y -185.018799,Z -337.307190,A 89.8236847,B 38.2151108,C -89.0491486,S 6,T 19,E1 0.0,E2 0.0,E3 0.0,E4 0.0,E5 0.0,E6 0.0}
DECL FDAT FP10={TOOL_NO 1,BASE_NO 2,IPO_FRAME #BASE,POINT2[] " ",TQ_STATE FALSE}
DECL E6POS XP410={X 570.135315,Y -87.9825745,Z -450.345490,A 87.9885483,B 38.2075691,C -88.4547653,S 6,T 19,E1 0.0,E2 0.0,E3 0.0,E4 0.0,E5 0.0,E6 0.0}
DECL FDAT FP410={TOOL_NO 1,BASE_NO 2,IPO_FRAME #BASE,POINT2[] " ",TQ_STATE FALSE}
DECL E6POS XP310={X 512.355347,Y -87.2580338,Z -650.326721,A 89.3334885,B 29.3791523,C -89.3156662,S 6,T 19,E1 0.0,E2 0.0,E3 0.0,E4 0.0,E5 0.0,E6 0.0}
DECL FDAT FP310={TOOL_NO 1,BASE_NO 2,IPO_FRAME #BASE,POINT2[] " ",TQ_STATE FALSE}
DECL E6POS XP210={X 512.274658,Y -74.7021561,Z -850.279,A 87.5055847,B 31.8261738,C -89.3899307,S 6,T 19,E1 0.0,E2 0.0,E3 0.0,E4 0.0,E5 0.0,E6 0.0}
DECL FDAT FP210={TOOL_NO 1,BASE_NO 2,IPO_FRAME #BASE,POINT2[] " ",TQ_STATE FALSE}
DECL E6POS XP110={X 542.657532,Y -70.7026291,Z -993.619934,A 88.1469650,B 31.7469406,C -88.1797943,S 6,T 19,E1 0.0,E2 0.0,E3 0.0,E4 0.0,E5 0.0,E6 0.0}
DECL FDAT FP110={TOOL_NO 1,BASE_NO 2,IPO_FRAME #BASE,POINT2[] " ",TQ_STATE FALSE}
DECL E6POS XP420={X 512.355347,Y -87.2580338,Z -650.326721,A 89.3334885,B 29.3791523,C -89.3156662,S 6,T 19,E1 0.0,E2 0.0,E3 0.0,E4 0.0,E5 0.0,E6 0.0}
DECL FDAT FP420={TOOL_NO 1,BASE_NO 2,IPO_FRAME #BASE,POINT2[] " ",TQ_STATE FALSE}
DECL E6POS XP320={X 512.274658,Y -74.7021561,Z -850.279,A 87.5055847,B 31.8261738,C -89.3899307,S 6,T 19,E1 0.0,E2 0.0,E3 0.0,E4 0.0,E5 0.0,E6 0.0}
DECL FDAT FP320={TOOL_NO 1,BASE_NO 2,IPO_FRAME #BASE,POINT2[] " ",TQ_STATE FALSE}
DECL E6POS XP220={X 542.657532,Y -70.7026291,Z -993.619934,A 88.1469650,B 31.7469406,C -88.1797943,S 6,T 19,E1 0.0,E2 0.0,E3 0.0,E4 0.0,E5 0.0,E6 0.0}
DECL FDAT FP220={TOOL_NO 1,BASE_NO 2,IPO_FRAME #BASE,POINT2[] " ",TQ_STATE FALSE}
DECL E6POS XP120={X 611.491638,Y -185.018967,Z -337.307312,A 89.8236847,B 38.2151108,C -89.0491562,S 6,T 19,E1 0.0,E2 0.0,E3 0.0,E4 0.0,E5 0.0,E6 0.0}
DECL FDAT FP120={TOOL_NO 1,BASE_NO 2,IPO_FRAME #BASE,POINT2[] " ",TQ_STATE FALSE}
DECL E6POS XP121={X 444.231262,Y 453.996155,Z 946.107,A -102.024231,B -19.0647125,C 118.088737,S 2,T 42,E1 0.0,E2 0.0,E3 0.0,E4 0.0,E5 0.0,E6 0.0}
DECL FDAT FP121={TOOL_NO 2,BASE_NO 1,IPO_FRAME #BASE,POINT2[] " ",TQ_STATE FALSE}
DECL E6POS XP_ABRIR10={X -388.316040,Y -25.2088261,Z 2663.06567,A 120.478897,B 28.0102959,C -44.0925598,S 2,T 11,E1 0.0,E2 0.0,E3 0.0,E4 0.0,E5 0.0,E6 0.0}
DECL FDAT FP_ABRIR10={TOOL_NO 9,BASE_NO 0,IPO_FRAME #BASE,POINT2[] " ",TQ_STATE FALSE}
DECL E6POS XP_AHOME={X 219.071762,Y 671.007507,Z 2930.63721,A 32.1725731,B 67.6234055,C -41.3866920,S 2,T 11,E1 0.0,E2 0.0,E3 0.0,E4 0.0,E5 0.0,E6 0.0}
DECL FDAT FP_aHOME={TOOL_NO 9,BASE_NO 0,IPO_FRAME #BASE,POINT2[] " ",TQ_STATE FALSE}
DECL E6POS XP11={X 500.256653,Y 161.434937,Z -226.642746,A -88.9033661,B 31.1327610,C 89.4967575,S 6,T 58,E1 0.0,E2 0.0,E3 0.0,E4 0.0,E5 0.0,E6 0.0}
DECL FDAT FP11={TOOL_NO 2,BASE_NO 1,IPO_FRAME #BASE,POINT2[] " ",TQ_STATE FALSE}
DECL E6POS XP0={X 549.337402,Y 294.945343,Z -525.939819,A -88.6139679,B 32.7546692,C 89.9199066,S 6,T 58,E1 0.0,E2 0.0,E3 0.0,E4 0.0,E5 0.0,E6 0.0}
DECL FDAT FP0={TOOL_NO 2,BASE_NO 1,IPO_FRAME #BASE,POINT2[] " ",TQ_STATE FALSE}
DECL LDAT LCPDAT1={VEL 2.00000,ACC 25.0000,APO_DIST 100.000,APO_FAC 50.0000,AXIS_VEL 100.000,AXIS_ACC 100.000,ORI_TYP #VAR,CIRC_TYP #BASE,JERK_FAC 50.0000,GEAR_JERK 50.0000,EXAX_IGN 0}
DECL PDAT PPDAT1={VEL 100.000,ACC 100.000,APO_DIST 100.000,GEAR_JERK 50.0000,EXAX_IGN 0}
DECL E6POS XP112211={X 548.096252,Y 56.0438080,Z -488.650848,A -88.5563202,B 27.2481651,C 89.8798828,S 6,T 58,E1 0.0,E2 0.0,E3 0.0,E4 0.0,E5 0.0,E6 0.0}
DECL FDAT FP112211={TOOL_NO 2,BASE_NO 1,IPO_FRAME #BASE,POINT2[] " ",TQ_STATE FALSE}
DECL PDAT PPDAT2={VEL 100.000,ACC 100.000,APO_DIST 100.000,GEAR_JERK 50.0000,EXAX_IGN 0}
DECL PDAT PPDAT3={VEL 100.000,ACC 100.000,APO_DIST 100.000,GEAR_JERK 50.0000,EXAX_IGN 0}
DECL PDAT PPDAT4={VEL 100.000,ACC 100.000,APO_DIST 100.000,GEAR_JERK 50.0000,EXAX_IGN 0}
DECL E6POS XP_FIN_ABRIR_B1={X 515.739929,Y 203.106186,Z -802.900696,A -88.4565048,B 31.1992207,C 90.3611603,S 6,T 58,E1 0.0,E2 0.0,E3 0.0,E4 0.0,E5 0.0,E6 0.0}
DECL FDAT FP_FIN_ABRIR_B1={TOOL_NO 2,BASE_NO 1,IPO_FRAME #BASE,POINT2[] " ",TQ_STATE FALSE}
DECL LDAT LH={VEL 2.00000,ACC 25.0000,APO_DIST 100.000,APO_FAC 50.0000,AXIS_VEL 100.000,AXIS_ACC 100.000,ORI_TYP #VAR,CIRC_TYP #BASE,JERK_FAC 50.0000,GEAR_JERK 50.0000,EXAX_IGN 0}
DECL E6POS XP1={X 107.474121,Y 230.481583,Z 2716.11304,A 164.879425,B -15.5853510,C 56.0520973,S 3,T 43,E1 0.0,E2 0.0,E3 0.0,E4 0.0,E5 0.0,E6 0.0}
DECL FDAT FP1={TOOL_NO 9,BASE_NO 0,IPO_FRAME #BASE,POINT2[] " ",TQ_STATE FALSE}
DECL PDAT PPDAT5={VEL 100.000,ACC 50.0000,APO_DIST 100.000,GEAR_JERK 50.0000,EXAX_IGN 0}
DECL E6POS XPOS_ESPERA_AREA2={X 107.474121,Y 230.481583,Z 2716.11304,A 68.9610901,B 57.3843727,C 3.65238047,S 3,T 11,E1 0.0,E2 0.0,E3 0.0,E4 0.0,E5 0.0,E6 0.0}
DECL FDAT FPOS_ESPERA_AREA2={TOOL_NO 9,BASE_NO 0,IPO_FRAME #BASE,POINT2[] " ",TQ_STATE FALSE}
DECL E6POS XPOS_AREA2_LIBRE={X -388.316,Y -25.2088432,Z 2663.06567,A 120.478897,B 28.0102959,C -44.0925598,S 2,T 11,E1 0.0,E2 0.0,E3 0.0,E4 0.0,E5 0.0,E6 0.0}
DECL FDAT FPOS_AREA2_LIBRE={TOOL_NO 9,BASE_NO 0,IPO_FRAME #BASE,POINT2[] " ",TQ_STATE FALSE}
DECL PDAT PPDAT6={VEL 100.000,ACC 100.000,APO_DIST 100.000,GEAR_JERK 50.0000,EXAX_IGN 0}
DECL E6POS XP2={X 583.941223,Y 445.536316,Z -649.569580,A 88.2479935,B 31.3274651,C -91.0029144,S 6,T 19,E1 0.0,E2 0.0,E3 0.0,E4 0.0,E5 0.0,E6 0.0}
DECL FDAT FP2={TOOL_NO 1,BASE_NO 2,IPO_FRAME #BASE,POINT2[] " ",TQ_STATE FALSE}
DECL LDAT LM={VEL 2.00000,ACC 35.0000,APO_DIST 25.0000,APO_FAC 50.0000,AXIS_VEL 100.000,AXIS_ACC 100.000,ORI_TYP #VAR,CIRC_TYP #BASE,JERK_FAC 50.0000,GEAR_JERK 50.0000,EXAX_IGN 0}
DECL E6POS XPOS_ESCAPE={X 607.684753,Y -557.686,Z -478.522552,A 89.8343506,B 38.2078819,C -89.0144424,S 6,T 19,E1 0.0,E2 0.0,E3 0.0,E4 0.0,E5 0.0,E6 0.0}
DECL FDAT FPOS_ESCAPE={TOOL_NO 2,BASE_NO 2,IPO_FRAME #BASE,POINT2[] " ",TQ_STATE FALSE}
DECL E6POS XP3={X 884.483948,Y 175.178665,Z -105.312004,A 87.2753067,B 0.382869542,C -89.4738388,S 6,T 19,E1 0.0,E2 0.0,E3 0.0,E4 0.0,E5 0.0,E6 0.0}
DECL FDAT FP3={TOOL_NO 1,BASE_NO 2,IPO_FRAME #BASE,POINT2[] " ",TQ_STATE FALSE}
DECL LDAT LM2={VEL 2.00000,ACC 35.0000,APO_DIST 100.000,APO_FAC 50.0000,AXIS_VEL 100.000,AXIS_ACC 100.000,ORI_TYP #VAR,CIRC_TYP #BASE,JERK_FAC 50.0000,GEAR_JERK 50.0000,EXAX_IGN 0}
DECL FDAT FAux_abrir_B5={TOOL_NO 1,BASE_NO 2,IPO_FRAME #BASE,POINT2[] " ",TQ_STATE FALSE}
DECL E6POS XP4={X 882.444,Y 184.281158,Z 82.5686188,A 88.2306137,B 8.74523449,C -89.2814636,S 6,T 19,E1 0.0,E2 0.0,E3 0.0,E4 0.0,E5 0.0,E6 0.0}
DECL FDAT FP4={TOOL_NO 1,BASE_NO 2,IPO_FRAME #BASE,POINT2[] " ",TQ_STATE FALSE}
DECL E6POS XP5={X 880.540283,Y 630.105774,Z 809.545410,A 92.2069550,B 25.3441467,C -87.7599640,S 6,T 51,E1 0.0,E2 0.0,E3 0.0,E4 0.0,E5 0.0,E6 0.0}
DECL FDAT FP5={TOOL_NO 1,BASE_NO 2,IPO_FRAME #BASE,POINT2[] " ",TQ_STATE FALSE}
DECL E6POS XPRAD={X 1423.00195,Y 124.794365,Z -184.368179,A 73.7225494,B 22.0144253,C -91.1981354,S 6,T 19,E1 0.0,E2 0.0,E3 0.0,E4 0.0,E5 0.0,E6 0.0}
DECL FDAT FPRAD={TOOL_NO 1,BASE_NO 2,IPO_FRAME #BASE,POINT2[] " ",TQ_STATE FALSE}
DECL PDAT PPDAT7={VEL 100.000,ACC 100.000,APO_DIST 100.000,GEAR_JERK 50.0000,EXAX_IGN 0}
DECL PDAT PPDAT8={VEL 100.000,ACC 100.000,APO_DIST 100.000,GEAR_JERK 50.0000,EXAX_IGN 0}
DECL E6POS XP6={X 458.358673,Y 175.066650,Z -421.589233,A 87.2811890,B 0.879289031,C -89.4738693,S 6,T 19,E1 0.0,E2 0.0,E3 0.0,E4 0.0,E5 0.0,E6 0.0}
DECL FDAT FP6={TOOL_NO 2,BASE_NO 2,IPO_FRAME #BASE,POINT2[] " ",TQ_STATE FALSE}
DECL LDAT LCPDAT2={VEL 2.00000,ACC 35.0000,APO_DIST 25.0000,APO_FAC 50.0000,AXIS_VEL 100.000,AXIS_ACC 100.000,ORI_TYP #VAR,CIRC_TYP #BASE,JERK_FAC 50.0000,GEAR_JERK 50.0000,EXAX_IGN 0}
DECL E6POS XP7={X 456.767517,Y 174.055176,Z -285.301117,A 87.2753067,B 0.382872403,C -89.4738464,S 6,T 19,E1 0.0,E2 0.0,E3 0.0,E4 0.0,E5 0.0,E6 0.0}
DECL FDAT FP7={TOOL_NO 2,BASE_NO 2,IPO_FRAME #BASE,POINT2[] " ",TQ_STATE FALSE}
DECL LDAT LCPDAT3={VEL 2.00000,ACC 35.0000,APO_DIST 25.0000,APO_FAC 50.0000,AXIS_VEL 100.000,AXIS_ACC 100.000,ORI_TYP #VAR,CIRC_TYP #BASE,JERK_FAC 50.0000,GEAR_JERK 50.0000,EXAX_IGN 0}
DECL E6POS XP8={X 455.487762,Y 156.997040,Z -95.3273239,A 88.2306,B 8.74523067,C -89.2815,S 6,T 19,E1 0.0,E2 0.0,E3 0.0,E4 0.0,E5 0.0,E6 0.0}
DECL FDAT FP8={TOOL_NO 2,BASE_NO 2,IPO_FRAME #BASE,POINT2[] " ",TQ_STATE FALSE}
DECL LDAT LCPDAT4={VEL 2.00000,ACC 35.0000,APO_DIST 25.0000,APO_FAC 50.0000,AXIS_VEL 100.000,AXIS_ACC 100.000,ORI_TYP #VAR,CIRC_TYP #BASE,JERK_FAC 50.0000,GEAR_JERK 50.0000,EXAX_IGN 0}
DECL E6POS XP9={X 453.993439,Y 241.984619,Z 326.782745,A 90.6163864,B 27.5276222,C -88.2672272,S 6,T 51,E1 0.0,E2 0.0,E3 0.0,E4 0.0,E5 0.0,E6 0.0}
DECL FDAT FP9={TOOL_NO 2,BASE_NO 2,IPO_FRAME #BASE,POINT2[] " ",TQ_STATE FALSE}
DECL LDAT LCPDAT5={VEL 2.00000,ACC 35.0000,APO_DIST 25.0000,APO_FAC 50.0000,AXIS_VEL 100.000,AXIS_ACC 100.000,ORI_TYP #VAR,CIRC_TYP #BASE,JERK_FAC 50.0000,GEAR_JERK 50.0000,EXAX_IGN 0}
DECL E6POS XP12={X 480.958588,Y 552.899841,Z 646.993408,A 92.2069626,B 25.3441410,C -87.7599411,S 6,T 51,E1 0.0,E2 0.0,E3 0.0,E4 0.0,E5 0.0,E6 0.0}
DECL FDAT FP12={TOOL_NO 2,BASE_NO 2,IPO_FRAME #BASE,POINT2[] " ",TQ_STATE FALSE}
DECL LDAT LCPDAT6={VEL 2.00000,ACC 35.0000,APO_DIST 25.0000,APO_FAC 50.0000,AXIS_VEL 100.000,AXIS_ACC 100.000,ORI_TYP #VAR,CIRC_TYP #BASE,JERK_FAC 50.0000,GEAR_JERK 50.0000,EXAX_IGN 0}
DECL E6POS XP13={X 481.539032,Y 554.072693,Z 687.970642,A 92.3442612,B 25.1508522,C -87.7190857,S 6,T 51,E1 0.0,E2 0.0,E3 0.0,E4 0.0,E5 0.0,E6 0.0}
DECL FDAT FP13={TOOL_NO 2,BASE_NO 2,IPO_FRAME #BASE,POINT2[] " ",TQ_STATE FALSE}
DECL LDAT LCPDAT7={VEL 2.00000,ACC 35.0000,APO_DIST 25.0000,APO_FAC 50.0000,AXIS_VEL 100.000,AXIS_ACC 100.000,ORI_TYP #VAR,CIRC_TYP #BASE,JERK_FAC 50.0000,GEAR_JERK 50.0000,EXAX_IGN 0}
ENDDAT
